INTERFACE ITestSuite EXTENDS __SYSTEM.IQueryInterface

METHOD ReRunTests
VAR_INPUT
END_VAR
END_METHOD

METHOD Test : ITestOperation
VAR_INPUT
	TestId : T_MaxString;
END_VAR
END_METHOD

END_INTERFACE

(* stored: Version 1.1.0.1
   Itf ITestSuite: Id {d78aa624-4cef-480e-b2e0-77b774c4b77c}
   Method ReRunTests: Id {cd5b05a7-7512-4eea-b6a2-26305dbec51d}
   Method Test: Id {42521a4e-2eec-4c69-8db8-d94d01afb442} *)
